FUNCTION TryConvert_BOOL_TO_DT : BOOL
VAR_INPUT
	in : BOOL;
	out : REFERENCE TO DT;
END_VAR

out := BOOL_TO_DT(in);
TryConvert_BOOL_TO_DT := TRUE;

END_FUNCTION

(* stored: Version 1.1.0.1, ProductVersion 3.1.4024.12
   POU TryConvert_BOOL_TO_DT: Id {2d17ef49-5710-4a6a-b436-c8dad875c819}, SpecialFunc None *)
